// TIA Portal V20 export
TYPE "typePhmi"
// stored: Access Published, IsFailsafeCompliant true, Namespace Safety
   STRUCT
      estop { ExternalWritable := 'False'} : Bool;   // Emergency Button
      enable { ExternalWritable := 'False'} : Bool;   // DeadMan Switch
      reset : Bool;
   END_STRUCT;
END_TYPE
